// SIMATIC STEP 7 (V5.x) project Q4
// CPU: CPU 313C
// station: Hardware
// station: SIMATIC 300(1)
// station: P_ADR_BUS
// program: S7 Program(1)

SYMBOL_TABLE
"Counter"	C 0	COUNTER
"Start"	I 0.0	BOOL
"Stop"	I 0.1	BOOL
"Reset"	I 0.2	BOOL
"L sensor"	I 0.3	BOOL
"M sensor"	I 0.4	BOOL
"Palletizing sensor"	I 0.5	BOOL
"Front limit-L"	I 0.7	BOOL
"Front limit-M"	I 1.1	BOOL
"Front limit-Pallet"	I 1.3	BOOL
"Emitter"	ID 30	DWORD
"Start/Stop mem"	M 0.0	BOOL
"P-memory"	M 0.1	BOOL
"M-memory"	M 0.2	BOOL
"L-memory"	M 0.3	BOOL
"P-count-memory"	M 0.4	BOOL
"M-count-memory"	M 0.5	BOOL
"L-count-memory"	M 0.6	BOOL
"On/Off Conveyor"	M 0.7	BOOL
"Pusher-L"	Q 0.3	BOOL
"Pusher-M"	Q 0.4	BOOL
"Pusher-Pallet"	Q 0.5	BOOL
"Conveyor"	Q 0.6	BOOL
"Start Button"	Q 0.7	BOOL
"Stop Button"	Q 1.0	BOOL
"Reset Button"	Q 1.1	BOOL
"CounterOut-L"	QD 30	DWORD
"CounterOut-M"	QD 34	DWORD
"CounterOut-Pallet"	QD 38	DWORD
END_SYMBOL_TABLE

ORGANIZATION_BLOCK OB 1
TITLE = "Main Program Sweep (Cycle)"
VERSION : 0.1
VAR_TEMP
  OB1_EV_CLASS : BYTE ;	//Bits 0-3 = 1 (Coming event), Bits 4-7 = 1 (Event class 1)
  OB1_SCAN_1 : BYTE ;	//1 (Cold restart scan 1 of OB 1), 3 (Scan 2-n of OB 1)
  OB1_PRIORITY : BYTE ;	//Priority of OB Execution
  OB1_OB_NUMBR : BYTE ;	//1 (Organization block 1, OB1)
  OB1_RESERVED_1 : BYTE ;	//Reserved for system
  OB1_RESERVED_2 : BYTE ;	//Reserved for system
  OB1_PREV_CYCLE : INT ;	//Cycle time of previous OB1 scan (milliseconds)
  OB1_MIN_CYCLE : INT ;	//Minimum cycle time of OB1 (milliseconds)
  OB1_MAX_CYCLE : INT ;	//Maximum cycle time of OB1 (milliseconds)
  OB1_DATE_TIME : DATE_AND_TIME ;	//Date and time OB1 started
END_VAR
BEGIN
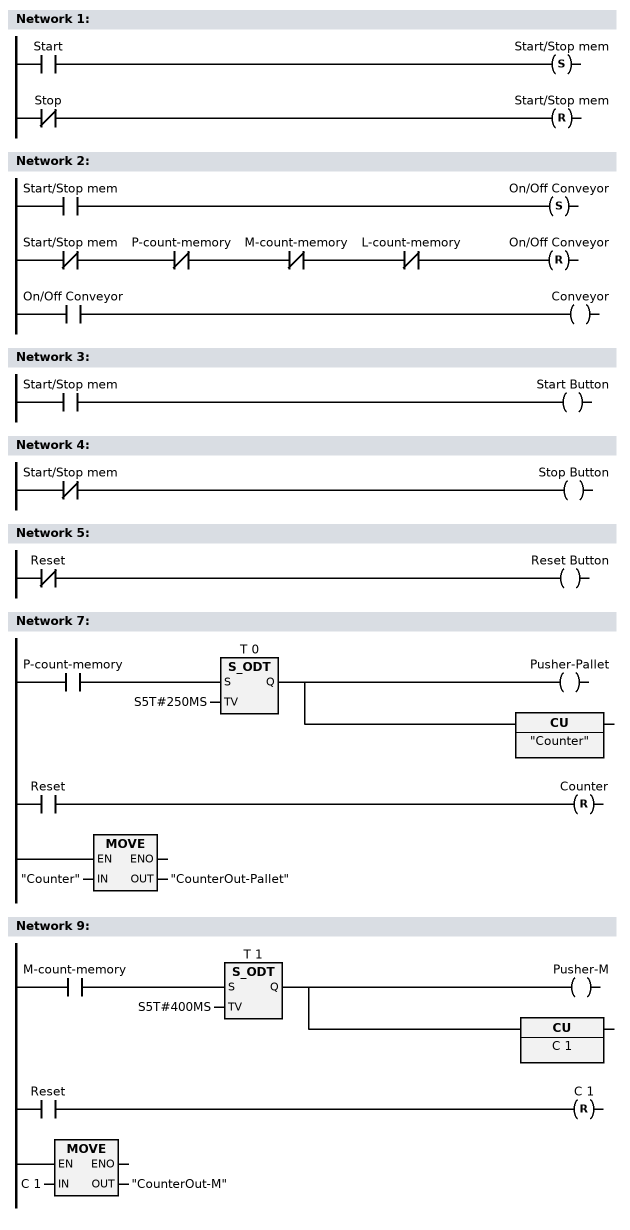
NETWORK
TITLE =
      A     "Start";
      S     "Start/Stop mem";
      AN    "Stop";
      R     "Start/Stop mem";
      NOP   0;
NETWORK
TITLE =
      A     "Start/Stop mem";
      S     "On/Off Conveyor";
      AN    "Start/Stop mem";
      AN    "P-count-memory";
      AN    "M-count-memory";
      AN    "L-count-memory";
      R     "On/Off Conveyor";
      A     "On/Off Conveyor";
      =     "Conveyor";
NETWORK
TITLE =
      A     "Start/Stop mem";
      =     "Start Button";
NETWORK
TITLE =
      AN    "Start/Stop mem";
      =     "Stop Button";
NETWORK
TITLE =
      AN    "Reset";
      =     "Reset Button";
NETWORK
TITLE =
      A(;
      A(;
      L     "Emitter";
      L     100;
      >I;
      );
      A(;
      L     "Emitter";
      L     140;
      <I;
      );
      S     "P-memory";
      A     "Front limit-Pallet";
      R     "P-memory";
      A     "P-memory";
      );
      A     "Palletizing sensor";
      S     "P-count-memory";
      A     "Front limit-Pallet";
      R     "P-count-memory";
      NOP   0;
NETWORK
TITLE =
      A     "P-count-memory";
      L     S5T#250MS;
      SD    T 0;
      NOP   0;
      NOP   0;
      NOP   0;
      A     T 0;
      =     L 20.0;
      A     L 20.0;
      BLD   102;
      =     "Pusher-Pallet";
      A     L 20.0;
      CU    "Counter";
      BLD   101;
      NOP   0;
      NOP   0;
      A     "Reset";
      R     "Counter";
      L     "Counter";
      T     "CounterOut-Pallet";
      NOP   0;
      NOP   0;
NETWORK
TITLE =
      A(;
      A(;
      L     "Emitter";
      L     170;
      >I;
      );
      A(;
      L     "Emitter";
      L     205;
      <I;
      );
      S     "M-memory";
      A     "Front limit-M";
      R     "M-memory";
      A     "M-memory";
      );
      A     "M sensor";
      S     "M-count-memory";
      A     "Front limit-M";
      R     "M-count-memory";
      NOP   0;
NETWORK
TITLE =
      A     "M-count-memory";
      L     S5T#400MS;
      SD    T 1;
      NOP   0;
      NOP   0;
      NOP   0;
      A     T 1;
      =     L 20.0;
      A     L 20.0;
      BLD   102;
      =     "Pusher-M";
      A     L 20.0;
      CU    C 1;
      BLD   101;
      NOP   0;
      NOP   0;
      A     "Reset";
      R     C 1;
      L     C 1;
      T     "CounterOut-M";
      NOP   0;
      NOP   0;
NETWORK
TITLE =
      A(;
      A(;
      L     "Emitter";
      L     210;
      >I;
      );
      S     "L-memory";
      A     "Front limit-L";
      R     "L-memory";
      A     "L-memory";
      );
      A     "L sensor";
      S     "L-count-memory";
      A     "Front limit-L";
      R     "L-count-memory";
      NOP   0;
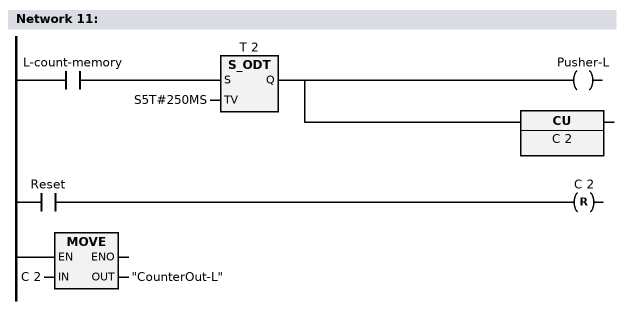
NETWORK
TITLE =
      A     "L-count-memory";
      L     S5T#250MS;
      SD    T 2;
      NOP   0;
      NOP   0;
      NOP   0;
      A     T 2;
      =     L 20.0;
      A     L 20.0;
      BLD   102;
      =     "Pusher-L";
      A     L 20.0;
      CU    C 2;
      BLD   101;
      NOP   0;
      NOP   0;
      A     "Reset";
      R     C 2;
      L     C 2;
      T     "CounterOut-L";
      NOP   0;
      NOP   0;
END_ORGANIZATION_BLOCK
